METHOD PUBLIC M_Run : BOOL
VAR_INPUT
	run:bool; // set to true to run, false to stop;
END_VAR

this^.iq_stPFO.pv_xRunSW := run;
END_METHOD

END_FUNCTION_BLOCK

// POUs/Functions/Valves/functions/F_RoughPumpInlet_ILK
(*
	Determine whether a pump attached to the inlet of a roughing pump is safe to open. 
	
	Return true, signaling it is safe to open when the roughing pump is confirmed to be working. 
*)

FUNCTION F_RoughPumpInlet_ILK : BOOL
VAR_INPUT
	ScrollPump	:	ST_RoughPump;
END_VAR
VAR
END_VAR


F_RoughPumpInlet_ILK := (ScrollPump.eState = pumpRUNNING); (* Confirm that the roughing pump is running before opening the valve *)

END_FUNCTION

// POUs/Functions/Valves/functions/F_TURBO_VRC_ILK
(* Close the vic if the roughing pump pirani loses its at-vac setpoint while the turbo is pumping *)
FUNCTION F_TURBO_VRC_ILK : BOOL
VAR_INPUT

	i_xHiVac 	: BOOL;
	i_xRunPTM	: BOOL;
	i_xFLVac	: BOOL;

END_VAR
VAR

	rHysterisis : REAL := 0;

	xInterlock: BOOL;
	rTolerance: REAL := 20;
END_VAR

(* Close the vic if the roughing pump pirani loses its at-vac setpoint while the turbo is pumping *)
F_TURBO_VRC_ILK := (NOT i_xHiVac AND NOT i_xRunPTM AND NOT i_xFLVac) OR
					(NOT i_xRunPTM AND i_xFLVac) OR
					(i_xRunPTM AND i_xFLVac);

END_FUNCTION

// POUs/Functions/Valves/functions/F_TurboGateValve_ILK
(* This Function Block evaluates the ILK condition of the Turbo Gate valve *)
(* The logic Protects the Turbo pump from inlet pressure above the SP*)

FUNCTION F_TurboGateValve_ILK : BOOL (* function return TRUE when ILK is OK*)
VAR_INPUT
	i_Turbo : ST_PTM; // Turbo Pump
	i_stISG : ST_VG; //Gauge measuring inlet Pressure e.g Pirani
END_VAR
VAR
END_VAR

(* This Function Block evaluates the ILK condition of the Turbo Gate valve *)
(* The logic Protects the Turbo pump from inlet pressure above the SP*)
F_TurboGateValve_ILK := (NOT (i_Turbo.eState = pumpSTOPPED) AND NOT (i_Turbo.eState = pumpSTOPPING) AND NOT (i_Turbo.eState = pumpFAULT))
						AND (i_stISG.xPRESS_OK AND i_stISG.rPRESS < i_Turbo.rInletPressureSP);

END_FUNCTION

// POUs/Functions/Valves/functions/F_TurboGateValve_ILK_1
(* This Function Block evaluates the ILK condition of the Turbo Gate valve *)
(* The logic Protects the Turbo pump from inlet pressure above the SP*)

FUNCTION F_TurboGateValve_ILK_1 : BOOL (* function return TRUE when ILK is OK*)
VAR_INPUT
	i_Turbo : ST_PTM; // Turbo Pump
	i_stISG : ST_VG; //Gauge measuring inlet Pressure e.g Pirani
END_VAR
VAR
END_VAR

(* This Function Block evaluates the ILK condition of the Turbo Gate valve *)
(* The logic Protects the Turbo pump from inlet pressure above the SP*)
F_TurboGateValve_ILK_1 := (NOT (i_Turbo.eState = pumpSTOPPED) AND NOT (i_Turbo.eState = pumpFAULT))
						AND (i_stISG.xPRESS_OK AND i_stISG.rPRESS < i_Turbo.rInletPressureSP);

END_FUNCTION

// POUs/Functions/Valves/functions/F_TurboGateValve_Protection_ILK
(* This Function Block evaluates the ILK condition of the Turbo Gate valve *)
(* The logic Protects the Turbo pump from inlet pressure above the SP*)
(* And Protects the Turbo pump from backing pressure above the SP*)
(* And Protects the Turbo pump in the case of backing pump not running*)

FUNCTION F_TurboGateValve_Protection_ILK : BOOL (* function return TRUE when ILK is OK*)
VAR_INPUT
	i_Turbo : ST_PTM; // Turbo Pump
	i_stISG : ST_VG; //Gauge measuring inlet Pressure e.g Pirani
	i_stBSG : ST_VG; //Gauge measuring backing Pressure e.g Pirani
	ScrollPump	:	ST_RoughPump; // Roughing pump
END_VAR
VAR
END_VAR

(* This Function Block evaluates the ILK condition of the Turbo Gate valve *)
(* The logic Protects the Turbo pump from inlet pressure above the SP*)
F_TurboGateValve_Protection_ILK := (NOT (i_Turbo.eState = pumpSTOPPED) AND NOT (i_Turbo.eState = pumpSTOPPING) AND NOT (i_Turbo.eState = pumpFAULT))
						AND (i_stISG.xPRESS_OK AND i_stISG.rPRESS < i_Turbo.rInletPressureSP)
						AND (i_stBSG.xPRESS_OK AND i_stBSG.rPRESS < i_Turbo.rBackingPressureSP)
						AND (ScrollPump.eState = pumpRUNNING);

END_FUNCTION

// POUs/Functions/Valves/functions/F_VALVE_REL_ILK
(* OK, this is going to be a general-use function that will return whether the ratio of the pressures given is less than x orders of magnitude.
True iff 10^(-x) < a/b < 10^x.  Simple, right?  Just make sure it gets a positive order of magnitude and the pressures aren't 0. ~Scott *)   
{attribute 'no_check'}
FUNCTION F_VALVE_REL_ILK : BOOL
VAR_INPUT
	i_stUSG	:	ST_VG; // Upstream Gague
	i_stDSG	:	ST_VG; // Downstream Gague
	//Orders of magnitude allowed between up/downstream pressures for valve to open. Must be real positive integer.
	i_iOrdersMagnitude: INT;
END_VAR
VAR
	rPressRatio : REAL;
	rMaxRatioAllowed	:	LREAL := EXPT(10,i_iOrdersMagnitude);
	rMinRatioAllowed	:	LREAL := EXPT(10,(-i_iOrdersMagnitude));
END_VAR

(* S. Stubbs 11/2015 *)

(* OK, this is going to be a general-use function that will return whether the ratio of the pressures given is less than x orders of magnitude.
True iff 10^(-x) < a/b < 10^x.  Simple, right?  Just make sure it gets a positive order of magnitude and the pressures aren't 0. ~Scott *)   

(* Find ratio *)

IF i_stDSG.rPRESS <> 0 THEN
	rPressRatio := i_stUSG.rPRESS / i_stDSG.rPRESS;

	F_VALVE_REL_ILK := rPressRatio < rMaxRatioAllowed AND rMinRatioAllowed < rPressRatio;
ELSE
	F_VALVE_REL_ILK := FALSE;
END_IF

END_FUNCTION

// POUs/Functions/Valves/functions/F_VRC_DIODE_ILK
(* The principle is simple, a VRC should never open when B side pressure is greater than 
the A side pressure. *)

FUNCTION F_VRC_DIODE_ILK : BOOL
VAR_INPUT

	i_stPGA : ST_VG; // A side pressure gauge
	i_stPGB	: ST_VG; // B side pressure gauge

END_VAR
VAR

	rHysterisis : REAL := 0;

	xInterlock: BOOL;
	rTolerance: REAL := 20;
END_VAR

(* The principle is simple, a VRC should never open when B side pressure is greater than the A side pressure. *)
rTolerance := 20;
F_VRC_DIODE_ILK := ((i_stPGA.rPRESS + rTolerance >= i_stPGB.rPRESS + rHysterisis) OR i_stPGA.xBAKEOUT) AND i_stPGA.xPRESS_OK AND i_stPGB.xPRESS_OK;

(* OK it gets a bit more complicated with hysterisis,

Now, if the F_VIC_DIODE_ILK is FALSE then some hysterisis is added to the B side. But if it's OK then we just stick with making sure that the A side is greater than the B side

*)
(*
IF NOT F_VIC_DIODE_ILK THEN
Hysterisis := 40;
ELSE
Hysterisis := 0;
END_IF
*)

END_FUNCTION

// POUs/Functions/Valves/functions/F_VRC_DIODE_ILK_OK
(*The function returns TRUE i.e. ILK_OK when pressure on A side is greater than or equal to the pressure on B side*)
FUNCTION F_VRC_DIODE_ILK_OK : BOOL
VAR_INPUT

	i_stPGA : ST_VG; // A side pressure gauge
	i_stPGB	: ST_VG; // B side pressure gauge

END_VAR
VAR
	rHysterisis : REAL := 0;

	xInterlock: BOOL;
	rTolerance: REAL := 0;
END_VAR

(* The principle is simple, a VRC should never open when B side pressure is greater than the A side pressure. *)
F_VRC_DIODE_ILK_OK := (i_stPGA.rPRESS + rTolerance >= i_stPGB.rPRESS + rHysterisis) AND i_stPGA.xPRESS_OK AND i_stPGB.xPRESS_OK;

END_FUNCTION

// POUs/Functions/Valves/Interfaces/FB_TVGC_ADS
(* This function block is created for interface devices between different PLC*)
(* Not all the fields in the original structure is required, just few signals *)
(*Use with FB_ADS_WATCHDOG on remotePLC*)
FUNCTION_BLOCK FB_TVGC_ADS extends FB_ADS
VAR_INPUT
	sNetId : String; //NetID of the Destination PLC controller
	nPort : UINT; // port number
	sVarName : string;// the variable name of the (device) declared function block.
	iWatchdog:UDINT;//The watchdog variable name written to by the remote plc
END_VAR
VAR_OUTPUT
	{attribute 'pytmc' := 'pv: '}
	VGC:ST_VGC;
	bError:BOOL;
END_VAR
VAR
	fb_CheckWatchdog: FB_CheckWatchdog;
	fb_Read_VGC: FB_ReadAdsSymByName;
	ftReset: F_TRIG;
	xFirstPass: bool:= true;
END_VAR

ftReset(CLK:= fb_Read_VGC.bBusy OR xFirstPass);
xFirstPass:=false;
(*calling ADS read function*)
fb_Read_VGC(
	bRead:= ftReset.Q, 
	sNetId:= sNetId, 
	nPort:= nPort, 
	sVarName:= CONCAT(sVarName,'.iq_stValve'), 
	nDestAddr:= ADR(VGC), 
	nLen:= SIZEOF(VGC), 
	tTimeout:= , 
	eComMode:= eAdsComModeFastCom, 
	bBusy=> , 
	bError=> , 
	nErrorId=> );
	

(*Error*)
fb_CheckWatchdog(
	bEnable:= TRUE, 
	tWatchdogTime:= T#900ms, 
	nCnt:= iWatchdog , 
	bWatchdog=> , 
	nLastCnt=> );
bError:= fb_Read_VGC.bError OR fb_CheckWatchdog.bWatchdog;

ACT_Logger();

ACTION ACT_Logger:
IF tErrorPresent.Q THEN
 IF(fb_Read_VGC.bError) THEN fbLogger(sMsg:='ADS Read Error', eSevr:=TcEventSeverity.Critical); END_IF;
 IF(fb_CheckWatchdog.bWatchdog) THEN fbLogger(sMsg:='ADS Watchdog Error', eSevr:=TcEventSeverity.Critical); END_IF;
END_IF
END_ACTION

END_FUNCTION_BLOCK

// POUs/Functions/Valves/Interfaces/FB_Valve_Interface
(* This function block is created for interface devices between different PLC*)
(* Not all the fields in the original structure is required, just few signals *)
(* They have to be linked to the custom created variables on the EL6692/5 primary side*)

FUNCTION_BLOCK FB_Valve_Interface
VAR_INPUT
END_VAR
VAR_OUTPUT
	{attribute 'pytmc' := 'pv: '}
	VGC:ST_VGC;
END_VAR
VAR
	i_xOpnLS AT%I*	: BOOL;
	i_xClsLS AT%I*	: BOOL;
END_VAR

(* This function block is created for interface devices between different PLC*)
(* Not all the fields in the original structure is required, just few signals *)
(* They have to be linked to the custom created variables on the EL6692/5 primary side*)


VGC.i_xClsLS := i_xClsLS;
VGC.i_xOpnLS := i_xOpnLS;

END_FUNCTION_BLOCK

// POUs/Functions/Valves/Interfaces/FB_VFS_Interface
(*Used as soft IO mapping to create a psuedo valve to communicate over two task on the same PLC.*) 
(*for FAST shutter control*)
FUNCTION_BLOCK FB_VFS_Interface EXTENDS FB_Valve
VAR_INPUT
	IG : ST_VG; // The MKS422 Cold Cathode Data Structure
END_VAR
VAR_OUTPUT
	{attribute 'pytmc' := '
    pv: ;
    '}
	iq_stValve : ST_VFS; (* All valve data and states will be in this struct*)
	i_xVAC_FAULT_OK AT%I*: BOOL; (*Valve Vacuum OK, is set to False when there is Vacuum Fault*)
END_VAR
VAR
	
	tonOvrd	:	TON;
	tOvrd	:	TIME := T#10s;
	(*outputs*)
	q_xPRESS_OK AT%Q*: BOOL;
	q_xOPN_SW AT%Q*:BOOL;
	q_xCLS_SW AT%Q*:BOOL; (*external open signal e.g epics*)
	q_xVAC_FAULT_Reset AT%Q*: BOOL; (*Valve Vacuum OK, is set to False when there is Vacuum Fault*)
	q_xOverrideMode AT%Q*: BOOL; (*To be linked to global override bit. This Overrides Vacuum logic only, EPS, MPS and PMPS are still enforces*)
	q_xOverrideOpen AT%Q*: BOOL;
	
	(*inputs*)
	i_xTrigger AT %I* : BOOL;
	i_xVFS_Open AT %I* : BOOL;
	i_xVFS_Closed AT %I* : BOOL;
	{attribute 'pytmc' := '
    pv: MPS_FAULT_OK
	field: ZNAM MPS FAULT ;
	field: ONAM MPS OK ;
	io: i ;
	'}
	i_xMPS_OK AT%I*: BOOL;(*MPS Fault OK, is set when the Valve is Open and there is no trigger*)
	i_eVFS_State AT%I*: E_VGC; (*Interface*)
END_VAR

(*soft IO Mapping*)

q_xPRESS_OK := IG.xPRESS_OK;

(* Soft IO Mapping*)
IO();
///Check valve postion
IF iq_stValve.i_xClsLS AND  iq_stValve.i_xOpnLS THEN
	iq_stValve.eState:=INVALID;
ELSIF NOT iq_stValve.i_xClsLS AND iq_stValve.i_xOpnLS THEN 
	iq_stValve.eState:=OPEN;
ELSIF iq_stValve.i_xClsLS AND NOT iq_stValve.i_xOpnLS THEN 
	iq_stValve.eState:=CLOSED;
ELSIF NOT iq_stValve.i_xClsLS AND NOT iq_stValve.i_xOpnLS THEN 
	iq_stValve.eState:=MOVING;
ELSE
	iq_stValve.eState:=INVALID;
END_IF
//Override timer
tonOvrd(IN:=q_xOverrideOpen, PT:=tOvrd);
(* Soft IO Mapping*)
IO();
(*Logger*)
ACT_Logger();

ACTION ACT_Logger:
// ILK logger

IF i_xTrigger AND ePrevState = OPEN THEN
 		fbLogger(sMsg:='Fast valve triggered to close', eSevr:=TcEventSeverity.Critical);  	
END_IF


//STATE Logger  

IF ePrevState <> iq_stValve.eState THEN
	  CASE iq_stValve.eState OF
		INVALID:
			fbLogger(sMsg:='Valve invalid position.', eSevr:=TcEventSeverity.Critical);
  		MOVING:
			fbLogger(sMsg:='Valve moving', eSevr:=TcEventSeverity.Warning);
		OPEN:
			fbLogger(sMsg:='Valve Open.', eSevr:=TcEventSeverity.Info);
		CLOSED:
			fbLogger(sMsg:='Valve closed.', eSevr:=TcEventSeverity.Info);
	  END_CASE
	  ePrevState := iq_stValve.eState;  
  END_IF
  


// Log valve timeouts
tErrorPresent(CLK:=iq_stValve.bErrorPresent);
IF tErrorPresent.Q THEN fbLogger(sMsg:=iq_stValve.sErrorMessage, eSevr:=TcEventSeverity.Warning); END_IF

// Log valve open
tAction(CLK:= iq_stValve.q_xOPN_DO);
IF tAction.Q THEN fbLogger(sMsg:='Valve commanded open', eSevr:=TcEventSeverity.Info); END_IF

// Log override mode enabled
tOverrideActivated(CLK:= (tonOvrd.Q AND q_xOverrideMode));
IF tOverrideActivated.Q THEN fbLogger(sMsg:='Valve override mode activated', eSevr:=TcEventSeverity.Warning); END_IF
END_ACTION

ACTION IO:
(*inputs*)
iq_stValve.i_xTrigger := i_xTrigger;
iq_stValve.i_xOpnLS := 	i_xVFS_Open;
iq_stValve.i_xClsLS:=	i_xVFS_Closed;
iq_stValve.eVGC_State := i_eVFS_State;
iq_stValve.i_xVAC_FAULT_OK:= i_xVAC_FAULT_OK;
(*output*)
q_xOPN_SW := iq_stValve.pv_xOPN_SW;
q_xCLS_SW:= iq_stValve.xCLS_SW;
q_xVAC_FAULT_Reset :=  iq_stValve.pv_xAlmRst;
q_xOverrideMode :=iq_stValve.xOverrideMode;
q_xOverrideOpen := iq_stValve.pv_xOvrdOpn ;
iq_stValve.sGFS := IG.sPath;

//reset the commands 
IF ( iq_stValve.i_xOpnLS) THEN iq_stValve.pv_xOPN_SW := FALSE; END_IF
IF ( iq_stValve.i_xClsLS) THEN iq_stValve.xCLS_SW := FALSE; END_IF
END_ACTION

END_FUNCTION_BLOCK

// POUs/Functions/Valves/Interfaces/ITF_Valve
INTERFACE ITF_Valve

END_INTERFACE

// POUs/Functions/Valves/FB_Kashiyama_VRC
(* Main Kashiyama gate valve permit to be open when:
		1. pump is NORMAL operating status, and
	    2. chamber pressure is below HighSP or pump is at LowSpeed state.
	it will close if chamber pressure is below than lowSP for 180s.	
*)
FUNCTION_BLOCK FB_Kashiyama_VRC
VAR_IN_OUT
	
END_VAR
VAR_OUTPUT
	{attribute 'pytmc' := ' pv:'}
	q_stValve : ST_VRC;
END_VAR
VAR_INPUT
	Pump : ST_KashiyamaDryPump;//Kashyiama pump
	i_xExtILK_OK : BOOL; //Connect to Interlock logic condition(e.g F_TURBO_VRC_ILK Function), otherwise, Set to True if the valve is not interlocked
	Gauge : ST_VG;// Pressure Gauge	
	i_xOverrideMode : BOOL;
END_VAR
VAR
	At_HiVac : BOOL;
	tmrTP : TP;
	tmrPT: TIME := T#180S;
	v1: BOOL;
	tonOvrd	:	TON;
	tonDelOK : TON;
	rtOK	:	R_TRIG;
	
	(*IO*)
	i_xOpnLS	AT%I*: BOOL;
	i_xClsLS	AT%I*: BOOL;
	q_xOPN_DO	AT%Q*: BOOL;
	
END_VAR

(* Main Kashiyama gate valve permit to be open when:
		1. pump is NORMAL operating status, and
	    2. chamber pressure is below HighSP or pump is at LowSpeed state.
	it will close if chamber pressure is below than lowSP for 60s.	
*)
(* 
      For main Kayshiyama pump's gate valve:
		Pump LowSP is MU100 base pressure (20 mTorr) 
		Pump HighSP is 600 Torr;
	  Second Kayshiyama pump allow Gas Attenuator operating at higher pressure, 
      it's gate valve is to be open when Gas Attenuator chamber pressure is above lowSP.  
*)


///Check valve postion
IF NOT q_stValve.i_xClsLS AND q_stValve.i_xOpnLS THEN 
	q_stValve.eState:=OPEN;
ELSIF q_stValve.i_xClsLS AND NOT q_stValve.i_xOpnLS THEN 
	q_stValve.eState:=CLOSED;
ELSIF NOT q_stValve.i_xClsLS AND NOT q_stValve.i_xOpnLS THEN 
	q_stValve.eState:=MOVING;
ELSE
	q_stValve.eState:=INVALID;
END_IF

//valve open interlock
q_stValve.xOPN_OK := Pump.i_xIsRun AND Pump.RdyTmr <= 0.0 AND (Gauge.rPRESS < Pump.HighSP OR Pump.q_xLspdDo) AND i_xExtILK_OK;
 

(* Override logic *)
(* Goal: give ability to override, but do so in a way that people won't forget it.
Solution: Override only after ten seconds of override, protect against blips,
when the valve permission goes true for more than ten seconds consistently, remove override
*)

tonDelOK(IN:=q_stValve.xOPN_OK, PT:=T#10S);
rtOK(CLK:=tonDelOK.Q);
IF rtOK.Q THEN q_stValve.pv_xOvrdOpn :=FALSE; END_IF

//Override timer
tonOvrd(IN:=q_stValve.pv_xOvrdOpn, PT:=T#10S);


(* Here's where the valve closes *)
IF NOT q_stValve.xOPN_OK AND NOT tonOvrd.Q THEN
q_stValve.pv_xOPN_SW := FALSE;
END_IF

At_HiVac := Gauge.xPRESS_OK AND Gauge.rPRESS < Pump.LowSP;
tmrTP (IN := At_HiVac AND q_stValve.q_xOPN_DO , PT := tmrPT);

IF At_HiVac AND q_stValve.q_xOPN_DO AND NOT tmrTP.Q THEN
	q_stValve.pv_xOPN_SW := FALSE ;
END_IF

(* Here's where the valve opens *)
q_stValve.q_xOPN_DO := (q_stValve.pv_xOPN_SW AND q_stValve.xOPN_OK) OR (tonOvrd.Q AND i_xOverrideMode); 

(*Soft IO Mapping*)
ACT_IO();

ACTION ACT_IO:
(*inputs*)
q_stValve.i_xOpnLS := 	i_xOpnLS;
q_stValve.i_xClsLS:=	i_xClsLS;
(*outputs*)
q_xOPN_DO:= q_stValve.q_xOPN_DO;
END_ACTION

END_FUNCTION_BLOCK

// POUs/Functions/Valves/FB_MKS248
(* MKS248 valve using MKS1249 Drive Module *)
FUNCTION_BLOCK FB_MKS248
VAR_INPUT
	i_xExtIlkOK	:	BOOL; //External Interlock, SET to TRUE if not used
	i_rReqPos	:	REAL; //Requested position
END_VAR
VAR_OUTPUT
	{attribute 'pytmc' := 'pv:'}
	iq_stVFN	:	ST_VCN; //Needle valve structure
END_VAR
VAR CONSTANT
	rOpenVoltage	:	REAL := 9.8; 
	rCloseVoltage	:	REAL := 0;	
END_VAR
VAR
	// Requested voltage
	rReqVoltage: REAL := 0;
	(*IO*)
	q_iRawPosition AT%Q* :INT;
END_VAR

(* MKS248 valve using MKS1249 Drive Module *)


// Interlocking
iq_stVFN.xIlkOK := i_xExtIlkOK;
(*Checking which Control mode is selected*)
IF iq_stVFN.xIlkOK THEN
	IF iq_stVFN.eValveControl = OpenValve THEN
		iq_stVFN.rReqPosition := iq_stVFN.rUpperLimit;(*Percentage*)// iq_stVCN.rUpperLimit;
	ELSIF iq_stVFN.eValveControl = CloseValve THEN
		iq_stVFN.rReqPosition := 0; (*Percentage*)
	ELSIF iq_stVFN.eValveControl = ManualControl THEN
		iq_stVFN.rReqPosition := LIMIT(0, iq_stVFN.rReqPosition, iq_stVFN.rUpperLimit);
	ELSIF iq_stVFN.eValveControl = PressureControl THEN
		iq_stVFN.rReqPosition := LIMIT(0, i_rReqPos, iq_stVFN.rUpperLimit); 
	END_IF
ELSE
	iq_stVFN.rReqPosition := 0;
	iq_stVFN.eValveControl := CloseValve;
END_IF

// Requested Voltage calculation
rReqVoltage := iq_stVFN.rReqPosition * (rOpenVoltage-rCloseVoltage)/100 + rCloseVoltage;
rReqVoltage := LIMIT(rCloseVoltage, rReqVoltage, rOpenVoltage); //The requested voltage should remain within this range
//Raw position calc
iq_stVFN.q_iRawPosition := REAL_TO_INT( 32767/10 * rReqVoltage);	
(*IO Mapping*)
ACT_IO();

ACTION ACT_IO:
(*outputs*)
q_iRawPosition := iq_stVFN.q_iRawPosition;
END_ACTION

END_FUNCTION_BLOCK

// POUs/Functions/Valves/FB_TurbVentvalve_NO
(* This function block impelemets Interlock for Agilent Turbo Vent Valve Normally Open*)
FUNCTION_BLOCK FB_TurbVentvalve_NO
VAR_OUTPUT
	{attribute 'pytmc' :=' pv:'}
	q_stValve : ST_VCC_NO;
END_VAR
VAR_INPUT
	i_stPTM	: ST_AgilentPTM; //Agilent Turbo Pump
END_VAR
VAR
	tofTmr 		: 	TOF;
	
	(*Output*)
	q_xCLS_DO AT%Q* : BOOL;
END_VAR

(*If the turbo is on, you cannot open the valve. In order to open the valve, you have to allow the turbopump
 to have already been turned off for 2 minutes and you have to press the open button on the vent valve

If the code looks confusing please use a truth table to verify*)

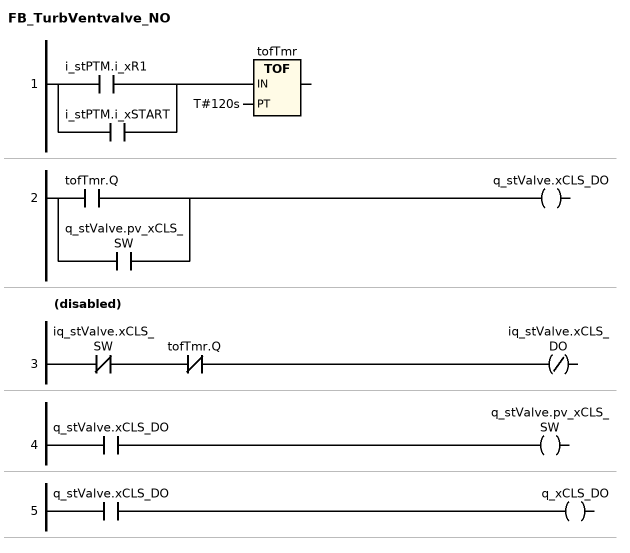
// NETWORK 1
tofTmr(IN := i_stPTM.i_xR1 OR i_stPTM.i_xSTART, PT := T#120s); // TOF

// NETWORK 2
q_stValve.xCLS_DO := tofTmr.Q OR q_stValve.pv_xCLS_SW;

// NETWORK 3 (disabled)
// iq_stValve.xCLS_DO := NOT (NOT iq_stValve.xCLS_SW AND NOT tofTmr.Q);

// NETWORK 4
q_stValve.pv_xCLS_SW := q_stValve.xCLS_DO;

// NETWORK 5
q_xCLS_DO := q_stValve.xCLS_DO;

ACTION ACT_IO:
(*outputs*)
q_xCLS_DO:= q_stValve.xCLS_DO;
END_ACTION

METHOD M_Close : BOOL
VAR_INPUT
		close:BOOL; //True to CLose, False to OPEN
END_VAR
This^.q_stValve.pv_xCLS_SW :=Close;
END_METHOD

END_FUNCTION_BLOCK

// POUs/Functions/Valves/FB_VCN
(* This function implements the Basic functions for the Pfeiffer EVR 116 needle valve*)
FUNCTION_BLOCK FB_VCN
VAR_INPUT
	i_xExtIlkOK	:	BOOL; //External Interlock, SET to TRUE if not used
	i_ReqPos	:	REAL; //Requested position

END_VAR
VAR_OUTPUT
	{attribute 'pytmc' := '
    pv:
	'}
	iq_stVCN	:	ST_VCN; //Needle valve structure
END_VAR
VAR_IN_OUT
	
END_VAR

VAR CONSTANT
	rOpenVoltage	:	REAL := 9.1; // From the EVR 116 manual, A Voltage of 9V it is completely Open
	rCloseVoltage	:	REAL := 0.4;// a voltage <0.5 V the valve is closed	
END_VAR
VAR
	// Requested voltage
	{attribute 'pytmc' := '
	pv: POS_AO;
	io: i ;
	'}
	rReqVoltage: REAL := 0;
	//iResolution: INT :=16;
	// 
	(*IO*)
	q_iRawPosition AT%Q* :INT;

END_VAR

(* Needle valve control FB
A. Wallace 2016-7-21

This FB should be used as a low level control block.

It provides:

Valve position ceiling
Interlock
Scaling

It is not intended for:
Closed-loop control

It could be used for:
Valve position/flow linearization

Note: Raw position calc is based on 0.5 to 9V span, 32767 bits
*)

// Interlocking
iq_stVCN.xIlkOK := i_xExtIlkOK;
(*Checking which Control mode is selected*)
IF iq_stVCN.xIlkOK THEN
	IF iq_stVCN.eValveControl = OpenValve THEN
		iq_stVCN.rReqPosition := iq_stVCN.rUpperLimit;(*Percentage*)// iq_stVCN.rUpperLimit;
	ELSIF iq_stVCN.eValveControl = CloseValve THEN
		iq_stVCN.rReqPosition := 0; (*Percentage*)
	ELSIF (iq_stVCN.eValveControl = ManualControl) (*AND (iq_stVCN.xOPN_SW)*) THEN
		iq_stVCN.rReqPosition := LIMIT(0, iq_stVCN.rReqPosition, iq_stVCN.rUpperLimit);
	ELSIF iq_stVCN.eValveControl = PressureControl THEN
		iq_stVCN.rReqPosition := LIMIT(0, i_ReqPos, iq_stVCN.rUpperLimit); 
	END_IF
ELSE
	iq_stVCN.rReqPosition := 0;
	iq_stVCN.eValveControl := CloseValve;
END_IF

// Requested Voltage calculation
rReqVoltage := iq_stVCN.rReqPosition * (rOpenVoltage-rCloseVoltage)/100 + rCloseVoltage;
rReqVoltage := LIMIT(rCloseVoltage, rReqVoltage, rOpenVoltage); //The requested voltage should remain within this range
//Raw position calc
iq_stvcn.q_iRawPosition := REAL_TO_INT( 32767/10 * rReqVoltage);	

(*SOft IO Mapping*)
ACT_IO();

ACTION ACT_IO:
(*outputs*)
q_iRawPosition := iq_stVCN.q_iRawPosition;
(*inputs*)
iq_stVCN.i_iPosition := iq_stvcn.q_iRawPosition;
END_ACTION

METHOD M_ValveControl : BOOL
VAR_INPUT
	state:E_VCN; // Close, Open, Pressure, Manual
END_VAR
iq_stVCN.eValveControl := state;
END_METHOD

END_FUNCTION_BLOCK

// POUs/Functions/Valves/FB_VFS
(* This function block implements basic functionality for Fast Shutter/Valves*)
(* Create a separate virtual PLC for the fast shutter logic, and tie/map this task to the FAST I/O portion of the ethercat bus,
 so we can scan these I/Os faster than the rest of the vacuum I/Os.
The Fast shutter was tested with PLC task Cycle Base Time 50us with cycle time 0.050ms.
*)
FUNCTION_BLOCK FB_VFS EXTENDS FB_Valve
VAR_INPUT
	i_xPMPS_OK:	BOOL	; (*External MPS interlock, Set to TRUE when no PMPS interlock is required*)
	i_xExt_OK: BOOL; (*Other External Interlock, Set to True when no external interlock is required*)
	i_sDevName : T_MaxString :=  'VGC'; // Device name for diagnostic
END_VAR
VAR_IN_OUT
	io_fbFFHWO    :    FB_HardwareFFOutput;
END_VAR
VAR
	xOPN_OK :BOOL;
	xERR_ExtFault :BOOL; 
	// PMPS
	fbFF    :    FB_FastFault :=(
        i_DevName := 'VFS',
        i_Desc := 'Fault occurs when fast valve is not in open state',
        i_TypeCode := 16#1010);
	
	rDiffPressAllowed	:	REAL := 22.5; // Torr, Default value comes from Vat Valve Manual
	rDiffPress : REAL;
	set : BOOL;
    reset: BOOL;
	  
	xFirstPass	:	BOOL := TRUE;
	//fbFSInit		:	R_TRIG;
	rtOPN_SW :	R_TRIG;
		
	tonDelOK : TON;
	rtOK	:	R_TRIG;
	tonOvrd	:	TON;
	
	tDelOK	:	TIME := T#60S;
	tOvrd	:	TIME := T#10s;
	
	xClose: BOOL;
	xOpen: BOOL;
	CloseTimer: TON;
	TimDur: TIME := T#20MS;
	OpenTimer: TON;
	OpenTimDur: TIME := T#2S;
	
	(* Timeouts*)
	tCLSTimeOutDuration: TIME:= T#0.5S;
	tOPNTimeOutDuration: TIME:= T#10S;
	tOPNtimeout: TON;
	tCLStimeout:TON;
	

	(*IO*)
	i_xOpnLS	AT%I*: BOOL;
	i_xClsLS	AT%I*: BOOL;
	q_xClose_A	AT%Q*: BOOL;
	q_xClose_B	AT%Q*: BOOL;
	q_xClose_C	AT%Q*: BOOL;
	q_xOPN_DO	AT%Q*: BOOL;
	i_xTrigger	AT%I*: BOOL; 
	
	// Interface
	i_xPress_OK AT%I*:BOOL; (*To be linked to the Fast sensor structure signal IG.xPRESS_OK, to make sure that the device is connected*)
	i_xOPN_SW AT%I*:BOOL;
	i_xCLS_SW AT%I*:BOOL; (*external open signal e.g epics*)
	i_xVAC_FAULT_Reset	AT%I*: BOOL;(*Valve Vacuum OK, is set to False when there is Vacuum Fault*)
	i_xOverrideMode AT%I*: BOOL; (*To be linked to global override bit. This Overrides Vacuum logic only, EPS, MPS and PMPS are still enforces*)
	i_xOverrideOpen AT%I*: BOOL;
	q_xTrigger	AT%Q*: BOOL; (*Interface*)
	q_xVFS_Open AT%Q*: BOOL; (*Interface*)
	q_xVFS_Closed AT%Q*: BOOL; (*Interface*)
	q_xVAC_FAULT_OK AT%Q*: BOOL; (*Valve Vacuum OK, is set to False when there is Vacuum Fault*)
	q_xMPS_OK	 AT%Q*:	BOOL; (*MPS Fault OK, is set when the Valve is Open and there is no trigger*)
	q_eVFS_State AT%Q*: E_VGC; (*Interface*)
	
END_VAR



(* Fast Shutter/Valve Function Block*)
(* M.Ghaly Feb 2019*)

(* Fast Shutters do not function as complete isolation valves, but are intended to rapidly limit conductance 
between vacuum regions.  They should be installed in conjunction with isolation gate valves.  The conductance 
of the fast shutter in the closed state may be sufficiently low as to create an isolated vacuum region.  
Thus, at least a pirani gauge, that can measure a pressure down to 1x10-4 Torr, needs to be installed between
the shutter and the isolation gate valve.
In the case where a gauge is not installed, the neigboring gate Valves should not be opened unless the shutter 
is Open. 
*)
(* On first PLC pass, put valve into vented state, which implies a closed valve *)
IF xFirstPass THEN
	fbFF.i_DevName := i_sDevName;
	xFirstPass := FALSE;
END_IF

(* Input Trigger to close the Fast Shutter*)
(* Neighboring Valves Should also be triggered to Close*)
IF (i_xTrigger) OR NOT (i_xPress_OK) OR NOT (i_xExt_OK)  OR i_xCLS_SW  THEN 
	xClose:= TRUE;
	xOpen:= FALSE;
	q_xVAC_FAULT_OK:= FALSE;
	IF (NOT i_xCLS_SW) THEN xERR_ExtFault := TRUE; END_IF;
	i_xCLS_SW := TRUE;
	q_xOPN_DO := FALSE;
	//i_xOPN_SW :=FALSE;
	xOpen:=FALSE;
ELSIF ((rtOPN_SW.Q) AND xOPN_OK AND NOT i_xOpnLS) OR (tonOvrd.Q AND i_xOverrideMode) THEN
	q_xOPN_DO := TRUE;
END_IF
IF (xClose) AND (NOT i_xClsLS) THEN
	q_xClose_A := TRUE;
	q_xClose_B := TRUE;
	q_xClose_C := TRUE;
END_IF
IF(CloseTimer.Q) OR (i_xClsLS) THEN
	q_xClose_A := FALSE;
	q_xClose_B := FALSE;
	q_xClose_C := FALSE;
	xClose := FALSE;
	//i_xOPN_SW := FALSE;
END_IF

IF(OpenTimer.Q) AND (i_xOpnLS) THEN
	q_xOPN_DO :=  FALSE;
	i_xOPN_SW := FALSE;
	xOpen:=FALSE;
END_IF

(* Neighboring Valves Interlock bit is reset When the Vacuum event error is reset and the Shutter is opened *)
IF (NOT i_xTrigger) AND (NOT xERR_ExtFault) AND i_xOpnLS THEN
	q_xVAC_FAULT_OK := TRUE;
END_IF

(*OPN OK evaluation bit *)
xOPN_OK := (NOT xERR_ExtFault) AND NOT i_xTrigger;

(* If Epics Command to close the Valve, check if PMPS, otherwise Keep command set to open valve *)
// is there really a PMPS requirment.



(* When the valve  is open MPS is OK*)
q_xMPS_OK := i_xOpnLS AND NOT i_xTrigger AND i_xPress_OK AND NOT(i_xCLS_SW);


(* Override logic *)
(* Goal: give ability to override, but do so in a way that people won't forget it.
Solution: Override only after ten seconds of override, protect against blips,
when the valve permission goes true for more than ten seconds consistently, remove override
*)

tonDelOK(IN:=xOPN_OK, PT:=tDelOK);
rtOK(CLK:=tonDelOK.Q);
IF rtOK.Q AND i_xOverrideOpen THEN 
	i_xOverrideOpen :=FALSE;
	//if (iq_stValve.eState = OPEN) AND (i_xOverrideMode) THEN iq_stValve.pv_xOPN_SW := TRUE; END_IF //for seamless transition   
    //Log
    fbLogger(sMsg:='Override expired', eSevr:=TcEventSeverity.Warning);
END_IF

//Override timer
tonOvrd(IN:=i_xOverrideOpen, PT:=tOvrd);


//Assign valve state
IF (i_xTrigger) THEN q_eVFS_State := E_VGC.Triggered;
ELSIF xERR_ExtFault THEN q_eVFS_State :=  E_VGC.Vac_Fault;
ELSIF NOT i_xClsLS AND tCLStimeout.Q THEN 
	q_eVFS_State :=  E_VGC.Cls_Timeout;
ELSIF NOT i_xOpnLS AND tOPNtimeout.Q THEN 
	q_eVFS_State :=  E_VGC.Opn_Timeout;
ELSE q_eVFS_State :=  E_VGC.At_Vac;
END_IF

(*Timers*)
CloseTimer ( IN:=xClose, PT:= TimDur, Q=>);
OpenTimer ( IN:=i_xOpnLS, PT:= OpenTimDur, Q=>);
tOPNtimeout(IN:= q_xOPN_DO, PT := tOPNTimeOutDuration);
tCLStimeout(IN:= q_xClose_A, PT := tCLSTimeOutDuration);
rtOPN_SW(CLK:= i_xOPN_SW);

(* Soft IO Mapping*)
IO();

(*Alarm reset *)
ACT_ResetAlarms();

(*FAST FAULT*)
fbFF(i_xOK := q_xMPS_OK,
    i_xReset := i_xVAC_FAULT_Reset,
	i_xAutoReset :=TRUE,
    io_fbFFHWO := io_fbFFHWO);

ACTION ACT_ResetAlarms:
//iq_stValve.xERR_DifPres R= i_xResetFault;

//iq_stValve.bErrorPresent R= i_xResetFault;

IF NOT i_xTrigger AND i_xPress_OK THEN
	xERR_ExtFault R= i_xVAC_FAULT_Reset;
	i_xVAC_FAULT_Reset:=FALSE;
END_IF
END_ACTION

ACTION IO:

q_xTrigger := i_xTrigger;
q_xVFS_Closed:= i_xClsLS;
q_xVFS_Open:= i_xOpnLS;
END_ACTION

END_FUNCTION_BLOCK

// POUs/Functions/Valves/FB_VRC
(* This Function Block Implements Basic Functionality for certain types of valves e.g Turbo Isolation valves, Apperture Valve.
This function block is interloked by an input (i_xExtILK_OK). This is so developers can interface with custom
interlocking logic outside this function block.*)
(* Note Interlock Logic is External *)
{attribute 'no_check'}
FUNCTION_BLOCK FB_VRC EXTENDS FB_Valve
VAR_IN_OUT
	
END_VAR
VAR_INPUT
	i_xExtILK_OK : BOOL; //Connect to Interlock logic condition(e.g F_TURBO_VRC_ILK Function), otherwise, Set to True if the valve is not interlocked
	i_xOverrideMode : BOOL; (*To be linked to global override bit. This Overrides Vacuum logic only, EPS, MPS and PMPS are still enforces*)
END_VAR
VAR_OUTPUT
	{attribute 'pytmc' := '
    pv:
	'}
	iq_stValve : ST_VRC;
END_VAR
VAR
	{attribute 'instance-path'}
	{attribute 'noinit'}
	sPath: STRING;
	xFirstPass	:	BOOL;
	fbFSInit		:	R_TRIG;
	tonOvrd	:	TON;
	tonDelOK : TON;
	rtOK	:	R_TRIG;
	tOvrd	:	TIME := T#10s;
	(* Timeouts*)
	tTimeOutDuration: TIME:= T#30S;
	tOPNtimeout: TON;
	tCLStimeout:TON;
	
	
	(*IO*)
	i_xOpnLS	AT%I*: BOOL;
	i_xClsLS	AT%I*: BOOL;
	q_xOPN_DO	AT%Q*: BOOL;

END_VAR


(* On first PLC pass, put valve into vented state, which implies a closed valve *)
fbFSInit( CLK := TRUE, Q => xFirstPass);
IF xFirstPass THEN
	iq_stValve.eVGC_State := Vented;
	iq_stValve.pv_xOPN_SW := FALSE;
	ePrevState := INVALID; 
END_IF




///Check valve position
IF iq_stValve.i_xClsLS AND  iq_stValve.i_xOpnLS THEN
	iq_stValve.eState:=INVALID;
ELSIF NOT iq_stValve.i_xClsLS AND iq_stValve.i_xOpnLS AND iq_stValve.q_xOPN_DO THEN 
	iq_stValve.eState:=OPEN;
ELSIF NOT iq_stValve.i_xClsLS AND iq_stValve.i_xOpnLS AND NOT iq_stValve.q_xOPN_DO THEN 
	iq_stValve.eState:=OPEN_F;
ELSIF iq_stValve.i_xClsLS AND NOT iq_stValve.i_xOpnLS AND NOT iq_stValve.q_xOPN_DO THEN 
	iq_stValve.eState:=CLOSED;
ELSIF NOT iq_stValve.i_xClsLS AND NOT iq_stValve.i_xOpnLS THEN 
	iq_stValve.eState:=MOVING;
ELSE
	iq_stValve.eState:=INVALID;
END_IF


(*evaluate Valve open external interlock*)
iq_stValve.xOPN_OK := i_xExtILK_OK;
iq_stValve.xEXT_OK := i_xExtILK_OK;
IF NOT iq_stValve.xOPN_OK and NOT tonOvrd.Q THEN
	iq_stValve.pv_xOPN_SW := FALSE;
	iq_stValve.eVGC_State := ERR_ExtFault;
END_IF

IF (iq_stValve.q_xOPN_DO) AND (iq_stValve.xOPN_OK) THEN
	iq_stValve.eVGC_State := AtVacuum;
END_IF
	

(* Override logic *)
(* Goal: give ability to override, but do so in a way that people won't forget it.
Solution: Override only after ten seconds of override, protect against blips,
when the valve permission goes true for more than ten seconds consistently, remove override
*)

tonDelOK(IN:=iq_stValve.xOPN_OK, PT:=T#10S);
rtOK(CLK:=tonDelOK.Q);
IF rtOK.Q AND iq_stValve.pv_xOvrdOpn THEN 
	iq_stValve.pv_xOvrdOpn :=FALSE; 
	if (iq_stValve.eState=OPEN) AND (i_xOverrideMode) THEN iq_stValve.pv_xOPN_SW := TRUE; END_IF
    //Log
    fbLogger(sMsg:='Override expired', eSevr:=TcEventSeverity.Warning);
END_IF
// Release the Force Open bit when the system override is false
IF NOT(i_xOverrideMode) THEN  iq_stValve.pv_xOvrdOpn :=FALSE; END_IF
//Override timer
tonOvrd(IN:=iq_stValve.pv_xOvrdOpn, PT:=tOvrd);

(* Here's where the valve opens *)
iq_stValve.q_xOPN_DO := (iq_stValve.pv_xOPN_SW AND iq_stValve.xOPN_OK) OR (tonOvrd.Q AND i_xOverrideMode);


///Check valve moving position timout
IF NOT iq_stValve.i_xClsLS AND tCLStimeout.Q THEN 
	iq_stValve.bErrorPresent := TRUE;
	iq_stValve.sErrorMessage := ' Close Timeout';
ELSIF NOT iq_stValve.i_xOpnLS AND tOPNtimeout.Q THEN 
	iq_stValve.bErrorPresent := TRUE; 
	iq_stValve.sErrorMessage := ' Open Timeout';
END_IF
IF (iq_stValve.eState=INVALID) THEN
	iq_stValve.bErrorPresent := TRUE; 
	iq_stValve.sErrorMessage := CONCAT(sPath,' Invalid Valve Position');
END_IF

(*Timers*)
tOPNtimeout(IN:= iq_stValve.q_xOPN_DO, PT := tTimeOutDuration );
tCLStimeout(IN:= NOT iq_stValve.q_xOPN_DO, PT := tTimeOutDuration);


(*Soft IO Mapping*)
ACT_IO();

// Log States and triggers
ACT_Logger();

ACTION ACT_IO:
(*inputs*)
iq_stValve.i_xOpnLS := 	i_xOpnLS;
iq_stValve.i_xClsLS:=	i_xClsLS;
iq_stValve.xOverrideMode := i_xOverrideMode;
(*outputs*)
q_xOPN_DO:= iq_stValve.q_xOPN_DO;
END_ACTION

ACTION ACT_Logger:
// ILK logger

IF NOT i_xExtILK_OK AND ePrevState = OPEN THEN
 		fbLogger(sMsg:='Lost external interlock while valve was open.', eSevr:=TcEventSeverity.Critical);  	
END_IF


//STATE Logger  

IF ePrevState <> iq_stValve.eState THEN
	  CASE iq_stValve.eState OF
		INVALID:
			fbLogger(sMsg:='Valve invalid position.', eSevr:=TcEventSeverity.Critical);
  		MOVING:
			fbLogger(sMsg:='Valve moving', eSevr:=TcEventSeverity.Warning);
		OPEN:
			fbLogger(sMsg:='Valve Open.', eSevr:=TcEventSeverity.Info);
		CLOSED:
			fbLogger(sMsg:='Valve closed.', eSevr:=TcEventSeverity.Info);
	  END_CASE
	  ePrevState := iq_stValve.eState;  
  END_IF
  


// Log valve timeouts
tErrorPresent(CLK:=iq_stValve.bErrorPresent);
IF tErrorPresent.Q THEN fbLogger(sMsg:=iq_stValve.sErrorMessage, eSevr:=TcEventSeverity.Warning); END_IF

// Log valve open
tAction(CLK:= iq_stValve.q_xOPN_DO);
IF tAction.Q THEN fbLogger(sMsg:='Valve commanded open', eSevr:=TcEventSeverity.Info); END_IF

// Log override mode enabled
tOverrideActivated(CLK:= (tonOvrd.Q AND i_xOverrideMode));
IF tOverrideActivated.Q THEN fbLogger(sMsg:='Valve override mode activated', eSevr:=TcEventSeverity.Warning); END_IF
END_ACTION

METHOD PUBLIC M_IsClosed : BOOL
VAR_INPUT
END_VAR
M_IsClosed := (This^.iq_stValve.eState = E_ValvePositionState.CLOSED);
END_METHOD

METHOD PUBLIC M_IsOpen : BOOL
VAR_INPUT
END_VAR
M_IsOpen := (This^.iq_stValve.eState = E_ValvePositionState.OPEN);
END_METHOD

// Use this Methode to Open or close the valve by setting the OPN_SW to the input value.
METHOD PUBLIC M_Set_OPN_SW : BOOL
VAR_INPUT
	value:BOOL;
END_VAR
This^.iq_stValve.pv_xOPN_SW := value;
END_METHOD

END_FUNCTION_BLOCK

// POUs/Functions/Valves/FB_VRC_EBD
(* This function block is similar to the FB_VGC, except it has 2 outputs to actuate the Valve*)
(* This Function Block Implements Basic Functionality for certain types of valves e.g Turbo Isolation valves, Apperture Valve *)
(* Note Interlock Logic is External *)
FUNCTION_BLOCK FB_VRC_EBD EXTENDS FB_Valve
VAR_IN_OUT
	
END_VAR
VAR_INPUT
	i_xExtILK_OK : BOOL; //Connect to Interlock logic condition(e.g F_TURBO_VRC_ILK Function), otherwise, Set to True if the valve is not interlocked
	i_xOverrideMode : BOOL; (*To be linked to global override bit. This Overrides Vacuum logic only, EPS, MPS and PMPS are still enforces*)
END_VAR
VAR_OUTPUT
	{attribute 'pytmc' := '
    pv:
	'}
	iq_stValve : ST_VRC;
END_VAR
VAR
	{attribute 'instance-path'}
	{attribute 'noinit'}
	sPath: STRING;
	xFirstPass	:	BOOL;
	fbFSInit		:	R_TRIG;
	tonOvrd	:	TON;
	tonDelOK : TON;
	rtOK	:	R_TRIG;
	tOvrd	:	TIME := T#10s;
	(* Timeouts*)
	tTimeOutDuration: TIME:= T#30S;
	tOPNtimeout: TON;
	tCLStimeout:TON;

	(*IO*)
	i_xOpnLS	AT%I*: BOOL;
	i_xClsLS	AT%I*: BOOL;
	q_xOPN_DO	AT%Q*: BOOL;
	q_xOPN_DO_2	AT%Q*: BOOL;
END_VAR


(* On first PLC pass, put valve into vented state, which implies a closed valve *)
fbFSInit( CLK := TRUE, Q => xFirstPass);
IF xFirstPass THEN
	iq_stValve.eVGC_State := Vented;
	iq_stValve.pv_xOPN_SW := FALSE;
END_IF


///Check valve position
IF NOT iq_stValve.i_xClsLS AND iq_stValve.i_xOpnLS THEN 
	iq_stValve.eState:=OPEN;
ELSIF iq_stValve.i_xClsLS AND NOT iq_stValve.i_xOpnLS THEN 
	iq_stValve.eState:=CLOSED;
ELSIF NOT iq_stValve.i_xClsLS AND NOT iq_stValve.i_xOpnLS THEN 
	iq_stValve.eState:=MOVING;
ELSE
	iq_stValve.eState:=INVALID;
END_IF

(*evaluate Valve open external interlock*)
iq_stValve.xOPN_OK := i_xExtILK_OK;
iq_stValve.xEXT_OK := i_xExtILK_OK;
IF NOT iq_stValve.xOPN_OK and NOT tonOvrd.Q THEN
	iq_stValve.pv_xOPN_SW := FALSE;
	iq_stValve.eVGC_State := ERR_ExtFault;
END_IF

IF (iq_stValve.q_xOPN_DO) AND (iq_stValve.xOPN_OK) THEN
	iq_stValve.eVGC_State := AtVacuum;
END_IF

(* Override logic *)
(* Goal: give ability to override, but do so in a way that people won't forget it.
Solution: Override only after ten seconds of override, protect against blips,
when the valve permission goes true for more than ten seconds consistently, remove override
*)

tonDelOK(IN:=iq_stValve.xOPN_OK, PT:=T#10S);
rtOK(CLK:=tonDelOK.Q);
IF rtOK.Q AND iq_stValve.pv_xOvrdOpn THEN 
	iq_stValve.pv_xOvrdOpn :=FALSE; 
	if (iq_stValve.eState=OPEN) AND (i_xOverrideMode) THEN iq_stValve.pv_xOPN_SW := TRUE; END_IF
    //Log
    fbLogger(sMsg:='Override expired', eSevr:=TcEventSeverity.Warning);
END_IF

//Override timer
tonOvrd(IN:=iq_stValve.pv_xOvrdOpn, PT:=T#10S);

(* Here's where the valve opens *)
iq_stValve.q_xOPN_DO := (iq_stValve.pv_xOPN_SW AND iq_stValve.xOPN_OK) OR (tonOvrd.Q AND i_xOverrideMode);

///Check valve moving postion timout
IF NOT iq_stValve.i_xClsLS AND tCLStimeout.Q THEN 
	iq_stValve.bErrorPresent := TRUE;
	iq_stValve.sErrorMessage := ' Close Timeout';
ELSIF NOT iq_stValve.i_xOpnLS AND tOPNtimeout.Q THEN 
	iq_stValve.bErrorPresent := TRUE; 
	iq_stValve.sErrorMessage := ' Open Timeout';
END_IF
IF (iq_stValve.eState=INVALID) THEN
	iq_stValve.bErrorPresent := TRUE; 
	iq_stValve.sErrorMessage := CONCAT(sPath,' Invalid Valve Position');
END_IF

(*Timers*)
tOPNtimeout(IN:= iq_stValve.q_xOPN_DO, PT := tTimeOutDuration );
tCLStimeout(IN:= NOT iq_stValve.q_xOPN_DO, PT := tTimeOutDuration);




(*Soft IO Mapping*)
ACT_IO();

// Log States and triggers
ACT_Logger();

ACTION ACT_IO:
(*inputs*)
iq_stValve.i_xOpnLS := 	i_xOpnLS;
iq_stValve.i_xClsLS:=	i_xClsLS;
iq_stValve.xOverrideMode := i_xOverrideMode;
(*outputs*)
q_xOPN_DO:= iq_stValve.q_xOPN_DO;
q_xOPN_DO_2:= iq_stValve.q_xOPN_DO;
END_ACTION

ACTION ACT_Logger:
// ILK logger

IF NOT i_xExtILK_OK AND ePrevState = OPEN THEN
 		fbLogger(sMsg:='Lost external interlock while valve was open.', eSevr:=TcEventSeverity.Critical);  	
END_IF


//STATE Logger  

IF ePrevState <> iq_stValve.eState THEN
	  CASE iq_stValve.eState OF
		INVALID:
			fbLogger(sMsg:='Valve invalid position.', eSevr:=TcEventSeverity.Critical);
  		MOVING:
			fbLogger(sMsg:='Valve moving', eSevr:=TcEventSeverity.Warning);
		OPEN:
			fbLogger(sMsg:='Valve Open.', eSevr:=TcEventSeverity.Info);
		CLOSED:
			fbLogger(sMsg:='Valve closed.', eSevr:=TcEventSeverity.Info);
	  END_CASE
	  ePrevState := iq_stValve.eState;  
  END_IF
  


// Log valve timeouts
tErrorPresent(CLK:=iq_stValve.bErrorPresent);
IF tErrorPresent.Q THEN fbLogger(sMsg:=iq_stValve.sErrorMessage, eSevr:=TcEventSeverity.Warning); END_IF

// Log valve open
tAction(CLK:= iq_stValve.q_xOPN_DO);
IF tAction.Q THEN fbLogger(sMsg:='Valve commanded open', eSevr:=TcEventSeverity.Info); END_IF

// Log override mode enabled
tOverrideActivated(CLK:= (tonOvrd.Q AND i_xOverrideMode));
IF tOverrideActivated.Q THEN fbLogger(sMsg:='Valve override mode activated', eSevr:=TcEventSeverity.Warning); END_IF
END_ACTION

METHOD PUBLIC M_IsClosed : BOOL
VAR_INPUT
END_VAR
M_IsClosed := (This^.iq_stValve.eState = E_ValvePositionState.CLOSED);
END_METHOD

METHOD PUBLIC M_IsOpen : BOOL
VAR_INPUT
END_VAR
M_IsOpen := (This^.iq_stValve.eState = E_ValvePositionState.OPEN);
END_METHOD

// Use this Methode to Open or close the valve by setting the OPN_SW to the input value.
METHOD PUBLIC M_Set_OPN_SW : BOOL
VAR_INPUT
	value:BOOL;
END_VAR
This^.iq_stValve.pv_xOPN_SW := value;
END_METHOD

END_FUNCTION_BLOCK

// POUs/Functions/Valves/FB_VRC_NO
(* This function block is different from the regular VRC in that CLOSING must be permitted. *)
FUNCTION_BLOCK FB_VRC_NO EXTENDS FB_Valve
VAR_IN_OUT

END_VAR
VAR_INPUT
	{attribute 'pytmc' := '
	pv: EXT_ILK_OK ;
	field: ZNAM NOT OK ;
	field: ONAM OK ;
	io: i ;
	'}
	i_xExtILK_OK : BOOL; //Connect to Interlock logic condition(e.g F_TURBO_VRC_ILK Function), otherwise, Set to True if the valve is not interlocked
	i_xOverrideMode : BOOL; (*To be linked to global override bit. This Overrides Vacuum logic only, EPS, MPS and PMPS are still enforces*)

END_VAR
VAR_OUTPUT
		iq_stValve : ST_VRC;
END_VAR
VAR

	{attribute 'noinit'}
	sPath: STRING;
	xFirstPass	:	BOOL;
	fbFSInit		:	R_TRIG;
	tonOvrd	:	TON;
	tonDelOK : TON;
	rtOK	:	R_TRIG;
	tOvrd	:	TIME := T#10s;
	(* Timeouts*)
	tTimeOutDuration: TIME:= T#30S;
	tOPNtimeout: TON;
	tCLStimeout:TON;
		{attribute 'pytmc' := '
	pv: CLS_SW ;
	field: ONAM CLOSE; 
	field: ZNAM OPEN;
	io: io ;
	'}
	pv_xCLS_SW	: BOOL;
	{attribute 'pytmc' := '
    pv: FORCE_CLS;
	io: io;
	'}
	pv_xOvrdCls	:	BOOL;

(*IO*)
	i_xOpnLS	AT%I*: BOOL;
	i_xClsLS	AT%I*: BOOL;
	q_xCLS_DO	AT%Q*: BOOL;

END_VAR

(* This function block is different from the regular VRC in that CLOSING must be permitted. *)

(* On first PLC pass, put valve into vented state, which implies a closed valve *)
fbFSInit( CLK := TRUE, Q => xFirstPass);
IF xFirstPass THEN
	pv_xCLS_SW := FALSE;
END_IF




///Check valve position
IF iq_stValve.i_xClsLS AND  iq_stValve.i_xOpnLS THEN
	iq_stValve.eState:=INVALID;
ELSIF NOT iq_stValve.i_xClsLS AND iq_stValve.i_xOpnLS AND iq_stValve.q_xOPN_DO THEN 
	iq_stValve.eState:=OPEN;
ELSIF iq_stValve.i_xClsLS AND NOT iq_stValve.i_xOpnLS AND NOT iq_stValve.q_xOPN_DO THEN 
	iq_stValve.eState:=CLOSED;
ELSIF NOT iq_stValve.i_xClsLS AND NOT iq_stValve.i_xOpnLS THEN 
	iq_stValve.eState:=MOVING;
ELSE
	iq_stValve.eState:=INVALID;
END_IF


(*evaluate Valve CLose external interlock*)
iq_stValve.xCLS_OK := i_xExtILK_OK;
IF NOT iq_stValve.xCLS_OK and NOT tonOvrd.Q THEN
	pv_xCLS_SW := FALSE;
END_IF


(* Override logic *)
(* Goal: give ability to override, but do so in a way that people won't forget it.
Solution: Override only after ten seconds of override, protect against blips,
when the valve permission goes true for more than ten seconds consistently, remove override
*)

tonDelOK(IN:=iq_stValve.xCLS_OK, PT:=T#10S);
rtOK(CLK:=tonDelOK.Q);
IF rtOK.Q AND pv_xOvrdCls THEN 
	pv_xOvrdCls :=FALSE; 
	if (iq_stValve.eState=CLOSED) AND (i_xOverrideMode) THEN pv_xCLS_SW := TRUE; END_IF
    //Log
    fbLogger(sMsg:='Override expired', eSevr:=TcEventSeverity.Warning);
END_IF

//Override timer
tonOvrd(IN:=pv_xOvrdCls, PT:=tOvrd);

(* Here's where the valve Actuates *)
q_xCLS_DO := ((iq_stValve.xCLS_OK  AND pv_xCLS_SW)OR (tonOvrd.Q AND i_xOverrideMode));
iq_stValve.q_xOPN_DO := NOT q_xCLS_DO;



///Check valve moving position timout
IF NOT iq_stValve.i_xClsLS AND tCLStimeout.Q THEN 
	iq_stValve.bErrorPresent := TRUE;
	//iq_stValve.sErrorMessage := ' Close Timeout';
ELSIF NOT iq_stValve.i_xOpnLS AND tOPNtimeout.Q THEN 
	iq_stValve.bErrorPresent := TRUE; 
	//iq_stValve.sErrorMessage := ' Open Timeout';
END_IF
IF (iq_stValve.eState=INVALID) THEN
	iq_stValve.bErrorPresent := TRUE; 
	//iq_stValve.sErrorMessage := CONCAT(sPath,' Invalid Valve Position');
END_IF

(*Timers*)
tOPNtimeout(IN:= iq_stValve.q_xOPN_DO, PT := tTimeOutDuration );
tCLStimeout(IN:= NOT iq_stValve.q_xOPN_DO, PT := tTimeOutDuration);


(*Soft IO Mapping*)
ACT_IO();

// Log States and triggers
ACT_Logger();

ACTION ACT_IO:
(*inputs*)
iq_stValve.i_xOpnLS := 	i_xOpnLS;
iq_stValve.i_xClsLS:=	i_xClsLS;
//iq_stValve. := i_xEXT_OK;
iq_stValve.xOverrideMode := i_xOverrideMode;
(*outputs*)
//q_xOPN_DO:= iq_stValve.q_xOPN_DO;
END_ACTION

METHOD PUBLIC M_IsClosed : BOOL
VAR_INPUT
END_VAR
M_IsClosed := (This^.iq_stValve.eState = E_ValvePositionState.CLOSED);
END_METHOD

METHOD PUBLIC M_IsOpen : BOOL
VAR_INPUT
END_VAR
M_IsOpen := (This^.iq_stValve.eState = E_ValvePositionState.OPEN);
END_METHOD

// Use this Methode to Open or close the valve by setting the OPN_SW to the input value.
METHOD PUBLIC M_Set_CLS_SW : BOOL
VAR_INPUT
		value:BOOL;
END_VAR
This^.pv_xCLS_SW := value;
END_METHOD

END_FUNCTION_BLOCK

// POUs/Functions/Valves/FB_VRC_OK_CLS
(* This function block is different from the regular VRC in that CLOSING must be permitted. *)
FUNCTION_BLOCK FB_VRC_OK_CLS
VAR_IN_OUT
	iq_stValve : ST_VRC;
END_VAR
VAR_INPUT
	i_xOverrideMode : BOOL;
END_VAR
VAR_OUTPUT
END_VAR
VAR

tonOvrd	:	TON;
tonDelOK : TON;
rtOK	:	R_TRIG;

END_VAR

(* This function block is different from the regular VRC in that CLOSING must be permitted. *)
(* Implemented for the funky valve 04 on LAMP *)
IF NOT iq_stValve.xOPN_OK and NOT tonOvrd.Q THEN
iq_stValve.pv_xOPN_SW := FALSE;
END_IF

(* Override logic *)
(* Goal: give ability to override, but do so in a way that people won't forget it.
Solution: Override only after ten seconds of override, protect against blips,
when the valve permission goes true for more than ten seconds consistently, remove override
*)

tonDelOK(IN:=iq_stValve.xOPN_OK, PT:=T#10S);
rtOK(CLK:=tonDelOK.Q);
IF rtOK.Q THEN iq_stValve.pv_xOvrdOpn :=FALSE; END_IF

//Override timer
tonOvrd(IN:=iq_stValve.pv_xOvrdOpn, PT:=T#10S);

(* Here's where the valve opens *)
iq_stValve.q_xOPN_DO := NOT iq_stValve.xCLS_OK OR ((iq_stValve.pv_xOPN_SW AND iq_stValve.xOPN_OK) OR (tonOvrd.Q AND i_xOverrideMode));

END_FUNCTION_BLOCK

// UnitTests/Functions/V_TO_INT
{attribute 'no_check'}
FUNCTION V_TO_INT : INT
VAR_INPUT
	analog : REAL;
END_VAR
VAR
	iBits :INT := 32767;
	iFullRange:INT := 10;
END_VAR

if ( iFullRange = 0 ) THEN iFullRange := 10;END_IF
V_TO_INT := REAL_TO_INT(analog * 32767 /iFullRange);

END_FUNCTION

// UnitTests/Gauges/FB_GCC_Test
FUNCTION_BLOCK FB_GCC_Test EXTENDS TcUnit.FB_TestSuite
VAR_INPUT
END_VAR
VAR_OUTPUT
END_VAR
VAR
	PG : ST_VG;
	fb_MKS422: FB_MKS422;
	//fb_MKS500: FB_MKS500;
	i_iPRESS_R AT %Q* :INT;
	cycle:INT :=0;
END_VAR

M_INIT();
M_Interlock();
M_CheckRange();
//M_SelfProtection();
cycle:=cycle+1;

METHOD M_CheckRange
VAR
	Expected:REAL;
	Actual:REAL;
	eStateExpected: E_PressureState;
	eStateActual: E_PressureState;
END_VAR
TEST('Check_Range');
Case This^.cycle of
	12:
	This^.i_iPRESS_R :=  V_TO_INT(0.61);
	This^.PG.rPRESS := 1E-4;
	This^.PG.xPRESS_OK := True;
	fb_MKS422.M_HVE(TRUE);
	
	15:
	TEST('MKS422_Range_937B');
	Expected :=1E-11 ;
	eStateExpected := Valid;
	Actual := This^.fb_MKS422.IG.rPRESS;
	eStateActual := This^.fb_MKS422.IG.eState;
	AssertTrue(This^.fb_MKS422.IG.xPRESS_OK, 'MKS422B xPRESS_OK is set to False');
	AssertEquals(eStateExpected,eStateActual,'MKS422B eState Fail');
	AssertEquals_REAL(Expected, Actual,1E-12, 'MKS422B rPress Fail');
	TEST_FINISHED_NAMED('MKS422_Range_937B');
	
	16:
	This^.i_iPRESS_R := V_TO_INT(2.4);
	This^.fb_MKS422.b937A:=TRUE;
	
	20:
	TEST('MKS422_Range_937A');
	Expected :=1E-8 ;
	Actual := This^.fb_MKS422.IG.rPRESS;
	eStateExpected := Valid;
	eStateActual := This^.fb_MKS422.IG.eState;
	AssertTrue(This^.fb_MKS422.IG.xPRESS_OK, 'MKS422A xPRESS_OK is set to False');
	AssertEquals(eStateExpected,eStateActual,'MKS422A eState Fail');
	AssertEquals_REAL(Expected, Actual,1E-9, 'MKS422A rPress Fail');
	TEST_FINISHED_NAMED('MKS422_Range_937A');

	
	21:
	This^.i_iPRESS_R :=  V_TO_INT(0.1);  
	
	
	24:
	TEST('MKS422_Range_Off');
	Expected :=0 ;
	eStateExpected := GaugeDisconnected;
	Actual := This^.fb_MKS422.IG.rPRESS;
	eStateActual := This^.fb_MKS422.IG.eState;
	AssertFalse(This^.fb_MKS422.IG.xPRESS_OK, 'MKS422A xPRESS_OK is set to True');
	AssertEquals(eStateExpected,eStateActual,'MKS422A eState Fail');
	AssertEquals_REAL(Expected, Actual,1, 'MKS422A rPress Fail');
	TEST_FINISHED_NAMED('MKS422_Range_Off');

	
	25:
	This^.i_iPRESS_R :=  V_TO_INT(10); 
	
	
	29:
	TEST('MKS422_Range_Invalid');
	Expected :=0 ;
	eStateExpected := PressInvalid;
	Actual := This^.fb_MKS422.IG.rPRESS;
	eStateActual := This^.fb_MKS422.IG.eState;
	AssertFalse(This^.fb_MKS422.IG.xPRESS_OK, 'MKS422A xPRESS_OK is set to True');
	AssertEquals(eStateExpected,eStateActual,'MKS422A eState Fail');
	AssertEquals_REAL(Expected, Actual,1, 'MKS422A rPress Fail');
	TEST_FINISHED_NAMED('MKS422_Range_Invalid');
	TEST_FINISHED_NAMED('Check_Range');

END_CASE

This^.fb_MKS422(PG:=This^.PG, IG=>);
END_METHOD

METHOD M_INIT
VAR
END_VAR
TEST('MKS422_Startup');
This^.PG.rPRESS := 1E-4;
This^.PG.xPRESS_OK := TRUE;
This^.fb_MKS422(PG:=This^.PG, IG=>);
IF( cycle = 3) THEN
	AssertFalse(This^.fb_MKS422.IG.xHV_SW, 'MKS422 xHV_SW set to True');
	AssertTrue(This^.fb_MKS422.IG.q_xHV_DIS, 'MKS422 q_xHV_DIS set to False');
	TEST_FINISHED_NAMED('MKS422_Startup');
End_IF;
END_METHOD

METHOD M_Interlock
VAR_INPUT
END_VAR
TEST('MKS422_Interlock_Active');
TEST('MKS422_Interlock_OK');
TEST('MKS422_Interlock_Lost');

Case cycle of
	1:
	This^.PG.rPRESS := 1E-1;
	This^.PG.xPRESS_OK := TRUE;
	fb_MKS422.M_HVE(TRUE);
	
	3:
	AssertFalse(This^.fb_MKS422.IG.xHV_SW, 'MKS422 xHV_SW set to True');
	AssertTrue(This^.fb_MKS422.IG.q_xHV_DIS, 'MKS422 q_xHV_DIS set to False');
	TEST_FINISHED_NAMED('MKS422_Interlock_Active');
	
	4:
	This^.PG.rPRESS := 1E-4;
	This^.PG.xPRESS_OK := True;
	fb_MKS422.M_HVE(TRUE);
	
	7:
	AssertTrue(This^.fb_MKS422.IG.xHV_SW, 'MKS422 xHV_SW set to False');
	AssertFalse(This^.fb_MKS422.IG.q_xHV_DIS, 'MKS422 q_xHV_DIS set to True');
	TEST_FINISHED_NAMED('MKS422_Interlock_OK');

	8:
	This^.PG.rPRESS := 1E-1;
	This^.PG.xPRESS_OK := False;
	This^.fb_MKS422(PG:=This^.PG, IG=>);
	
	11:
	AssertFalse(This^.fb_MKS422.IG.xHV_SW, 'MKS422 xHV_SW set to True');
	AssertTrue(This^.fb_MKS422.IG.q_xHV_DIS, 'MKS422 q_xHV_DIS set to False');
	TEST_FINISHED_NAMED('MKS422_Interlock_Lost');
END_CASE

This^.fb_MKS422(PG:=This^.PG, IG=>);
END_METHOD

METHOD M_SelfProtection
VAR_INPUT
END_VAR
// Switching the Cold cathode backon
TEST('MKS422_Interlock_OK_1');
This^.PG.rPRESS := 1E-4;
This^.PG.xPRESS_OK := True;
fb_MKS422.M_HVE(TRUE);
This^.fb_MKS422(PG:=This^.PG, IG=>);
AssertTrue(This^.fb_MKS422.IG.xHV_SW, 'MKS422 xHV_SW set to False');
AssertFalse(This^.fb_MKS422.IG.q_xHV_DIS, 'MKS422 q_xHV_DIS set to True');
TEST_FINISHED_NAMED('MKS422_Interlock_OK_1');

TEST('MKS422_Self_Protection');
This^.PG.rPRESS := 1E-3;
This^.PG.xPRESS_OK := TRUE;
This^.fb_MKS422(PG:=This^.PG, IG=>);
AssertFalse(This^.fb_MKS422.IG.xHV_SW, 'MKS422 xHV_SW set to True');
AssertTrue(This^.fb_MKS422.IG.q_xHV_DIS, 'MKS422 q_xHV_DIS set to False');
TEST_FINISHED_NAMED('MKS422_Self_Protection');
END_METHOD

END_FUNCTION_BLOCK

// UnitTests/Gauges/FB_GPI_Test
FUNCTION_BLOCK FB_GPI_Test EXTENDS TcUnit.FB_TestSuite
VAR_INPUT
END_VAR
VAR_OUTPUT
END_VAR
VAR
	fb_MKS275: FB_MKS275;
	fb_MKS317: FB_MKS317;
	i_iPRESS_R AT %Q* :INT;
	cycle:INT :=0;
END_VAR

M_INIT();
M_CheckRange();
cycle:=cycle+1;

METHOD M_CheckRange
VAR
	Expected:REAL;
	Actual:REAL;
	eStateExpected: E_PressureState;
	eStateActual: E_PressureState;
END_VAR

TEST('MKS275_Check_Range');
Case cycle of
	4:
	This^.i_iPRESS_R := V_TO_INT(3.674);
	Expected :=5 ;
	eStateExpected := Valid;
	
	7:
	TEST('MKS275_Range_R2');
	Actual := This^.fb_MKS275.PG.rPRESS;
	eStateActual := This^.fb_MKS275.PG.eState;
	AssertTrue(This^.fb_MKS275.PG.xPRESS_OK, 'MKS275 xPRESS_OK is set to False');
	AssertEquals(eStateExpected,eStateActual,'MKS275 eState Fail');
	AssertEquals_REAL(Expected, Actual,0.1, 'MKS275 rPress Fail');
	TEST_FINISHED_NAMED('MKS275_Range_R2');
	
	8:
	This^.i_iPRESS_R := V_TO_INT(5.614);
	Expected :=900 ;
	eStateExpected := Valid;
	
	
	12:
	TEST('MKS275_Range_R3');
	Actual := This^.fb_MKS275.PG.rPRESS;
	eStateActual := This^.fb_MKS275.PG.eState;
	AssertTrue(This^.fb_MKS275.PG.xPRESS_OK, 'MKS275 xPRESS_OK is set to False');
	AssertEquals(eStateExpected,eStateActual,'MKS275 eState Fail');
	AssertEquals_REAL(Expected, Actual,1, 'MKS275 rPress Fail');
	TEST_FINISHED_NAMED('MKS275_Range_R3');

	
	13:
	This^.i_iPRESS_R := V_TO_INT(0.3);
	Expected :=-1 ;
	eStateExpected := GaugeDisconnected;
	
	17:
	TEST('MKS275_Range_Off');
	Actual := This^.fb_MKS275.PG.rPRESS;
	eStateActual := This^.fb_MKS275.PG.eState;
	AssertTrue(This^.fb_MKS275.PG.xPRESS_OK, 'MKS275 xPRESS_OK is set to False');
	AssertEquals(eStateExpected,eStateActual,'MKS275 eState Fail');
	AssertEquals_REAL(Expected, Actual,1, 'MKS275 rPress Fail');
	TEST_FINISHED_NAMED('MKS275_Range_Off');

	
	18:
	This^.i_iPRESS_R := V_TO_INT(5.66);
	Expected :=-1 ;
	eStateExpected := OoR;
	
	22:
	TEST('MKS275_Range_OoR');
	Actual := This^.fb_MKS275.PG.rPRESS;
	eStateActual := This^.fb_MKS275.PG.eState;
	AssertTrue(This^.fb_MKS275.PG.xPRESS_OK, 'MKS275 xPRESS_OK is set to False');
	AssertEquals(eStateExpected,eStateActual,'MKS275 eState Fail');
	AssertEquals_REAL(Expected, Actual,1, 'MKS275 rPress Fail');
	TEST_FINISHED_NAMED('MKS275_Range_OoR');
	TEST_FINISHED_NAMED('MKS275_Check_Range');
	
END_CASE

This^.fb_MKS275(PG=>);
This^.fb_MKS317(PG=>);
END_METHOD

METHOD M_INIT
VAR
	Expected:REAL;
	Actual:REAL;
	eStateExpected: E_PressureState;
	eStateActual: E_PressureState;
END_VAR
// Start the Test
TEST('MKS275_Startup');
//Assign Voltage to FB
This^.i_iPRESS_R := V_TO_INT(0.384);
// Assigne expected result corresponing to the test input
Expected :=0.001 ;
eStateExpected := Valid;
//Instantiate the function block
This^.fb_MKS275(PG=>);
// Wait for few cycles 
IF( cycle = 3) THEN
	// Check the results
	Actual := This^.fb_MKS275.PG.rPRESS;
	eStateActual := This^.fb_MKS275.PG.eState;
	AssertTrue(This^.fb_MKS275.PG.xPRESS_OK, 'MKS275 xPRESS_OK is set to False');
	AssertEquals(eStateExpected,eStateActual,'MKS275 eState Fail');
	AssertEquals_REAL(Expected, Actual,0.0001, 'MKS275 rPress Fail');
	TEST_FINISHED_NAMED('MKS275_Startup');
END_IF
END_METHOD

END_FUNCTION_BLOCK

// UnitTests/Pumps/FB_PIP_Test
FUNCTION_BLOCK FB_PIP_Test EXTENDS TcUnit.FB_TestSuite
VAR_INPUT
END_VAR
VAR_OUTPUT
END_VAR
VAR
	PG : ST_VG;
	fb_PIP_GAMMA: FB_PIP_GAMMA;
END_VAR

M_INIT();
M_Interlock();
M_AutoStart();

METHOD M_AutoStart
VAR_INPUT
END_VAR
TEST('PIP_Auto_Restart');
This^.PG.rPRESS := 1E-6;
This^.PG.xPRESS_OK := TRUE;
This^.fb_PIP_GAMMA(i_stGauge:=PG, stPump=>, q_IG=>);
AssertTrue(This^.fb_PIP_GAMMA.stPump.q_xHVEna_DO, 'PIP HVEna_DO set to false');
TEST_FINISHED_NAMED('PIP_Auto_Restart');
END_METHOD

METHOD M_Check_State
VAR_INPUT
END_VAR
END_METHOD

METHOD M_INIT
VAR_INPUT
END_VAR
TEST('PIP_Startup');
This^.PG.rPRESS := 1E-1;
This^.PG.xPRESS_OK := TRUE;
This^.fb_PIP_GAMMA(i_stGauge:=PG, stPump=>, q_IG=>);
AssertFalse(This^.fb_PIP_GAMMA.stPump.xHVEna_SW, 'PIP xHVEna_SW set to True');
AssertFalse(This^.fb_PIP_GAMMA.stPump.q_xHVEna_DO, 'PIP HVEna_DO set to True');
TEST_FINISHED_NAMED('PIP_Startup');
END_METHOD

METHOD M_Interlock
VAR_INPUT
END_VAR
TEST('PIP_Interlock_Active');
This^.PG.rPRESS := 1E-1;
This^.PG.xPRESS_OK := True;
This^.fb_PIP_GAMMA.M_Run(TRUE);
This^.fb_PIP_GAMMA(i_stGauge:=PG, stPump=>, q_IG=>);
AssertFalse(This^.fb_PIP_GAMMA.stPump.xHVEna_SW, 'PIP xHVEna_SW set to True');
AssertFalse(This^.fb_PIP_GAMMA.stPump.q_xHVEna_DO, 'PIP HVEna_DO set to True');
TEST_FINISHED_NAMED('PIP_Interlock_Active');

TEST('PIP_Interlock_OK');
This^.PG.rPRESS := 1E-9;
This^.PG.xPRESS_OK := True;
This^.fb_PIP_GAMMA.M_Run(TRUE);
This^.fb_PIP_GAMMA(i_stGauge:=PG, stPump=>, q_IG=>);
AssertTrue(This^.fb_PIP_GAMMA.stPump.xHVEna_SW, 'PIP xHVEna_SW set to False');
AssertTrue(This^.fb_PIP_GAMMA.stPump.q_xHVEna_DO, 'PIP HVEna_DO set to False');
TEST_FINISHED_NAMED('PIP_Interlock_OK');

TEST('PIP_Interlock_Lost');
This^.PG.rPRESS := 1E-9;
This^.PG.xPRESS_OK := False;
This^.fb_PIP_GAMMA(i_stGauge:=PG, stPump=>, q_IG=>);
AssertFalse(This^.fb_PIP_GAMMA.stPump.xHVEna_SW, 'PIP xHVEna_SW set to True');
AssertFalse(This^.fb_PIP_GAMMA.stPump.q_xHVEna_DO, 'PIP HVEna_DO set to True');
TEST_FINISHED_NAMED('PIP_Interlock_Lost');
END_METHOD

END_FUNCTION_BLOCK

// UnitTests/Pumps/FB_PTM_Test
FUNCTION_BLOCK FB_PTM_Test EXTENDS TcUnit.FB_TestSuite
VAR_INPUT
END_VAR
VAR_OUTPUT
END_VAR
VAR
	fb_TwisTorr: FB_PTM_TwisTorr;
	fb_PTM_Ebara_010M:FB_PTM_Ebara_010M;
	
	cycle:INT :=0;
	(*IO*)
	q_iSpeedSet AT %I* :INT;
	i_diCurSpd AT %Q* :INT;
	
	i_iRawSpeed AT %Q* : INT; // Link to Analog input
	i_iTempMon AT %Q* : INT; // Link to Analog input -- input Voltage according to the pump temprature 0->5V 0->100C
	i_iCurrentMon AT %Q* : INT; //Link to Analog -- input Voltage to the output current of motor 0->5V 0->10A
	
END_VAR

M_INIT();
M_Interlock();
M_PTM_EBARA();
cycle:=cycle+1;

METHOD M_INIT : BOOL
VAR_INPUT
END_VAR
TEST('PTM_Twistorr_Startup');
fb_TwisTorr(i_xExtILKOk:= TRUE , iq_stPtm=> );
IF( cycle = 3) THEN
	AssertFalse(fb_TwisTorr.iq_stPtm.xRunSW ,'PTM Twistorr xRunSW is set to true');	
	AssertFalse(fb_TwisTorr.iq_stPtm.q_RunDO ,'PTM Twistorr q_RunDO is set to true');
	TEST_FINISHED_NAMED('PTM_Twistorr_Startup');
END_IF


TEST('PTM_Ebara011M_Startup');
fb_PTM_Ebara_010M(i_xExtILKOk:= TRUE , iq_stPtm=> );
IF( cycle = 3) THEN
	AssertFalse(fb_PTM_Ebara_010M.iq_stPtm.xRunSW ,'PTM Ebara011M xRunSW is set to true');	
	AssertFalse(fb_PTM_Ebara_010M.iq_stPtm.q_RunDO ,'PTM Ebara011M q_RunDO is set to true');
	AssertFalse(fb_PTM_Ebara_010M.iq_stPtm.q_xProtection ,'PTM Ebara011M q_xProtection is set to True');
	TEST_FINISHED_NAMED('PTM_Ebara011M_Startup');
END_IF
END_METHOD

METHOD M_Interlock
VAR_INPUT
END_VAR
TEST('PTM_Twistorr_Interlock_Active');
fb_TwisTorr.M_Run(TRUE);
fb_TwisTorr(i_xExtILKOk:= FALSE , iq_stPtm=> );
IF( cycle = 3) THEN
	AssertFalse(fb_TwisTorr.iq_stPtm.xRunSW ,'PTM Twistorr xRunSW is set to true');	
	AssertFalse(fb_TwisTorr.iq_stPtm.q_RunDO ,'PTM Twistorr q_RunDO is set to true');
	TEST_FINISHED_NAMED('PTM_Twistorr_Interlock_Active');
END_IF

TEST('PTM_Twistorr_Interlock_OK');
fb_TwisTorr.M_Run(TRUE);
fb_TwisTorr(i_xExtILKOk:= TRUE , iq_stPtm=> );
IF( cycle = 3) THEN
	AssertTrue(fb_TwisTorr.iq_stPtm.xRunSW ,'PTM Twistorr xRunSW is set to False');	
	AssertTrue(fb_TwisTorr.iq_stPtm.q_RunDO ,'PTM Twistorr q_RunDO is set to False');
	TEST_FINISHED_NAMED('PTM_Twistorr_Interlock_OK');
END_IF

TEST('PTM_Twistorr_Interlock_Lost');
fb_TwisTorr(i_xExtILKOk:= FALSE , iq_stPtm=> );
IF( cycle = 3) THEN
	AssertFalse(fb_TwisTorr.iq_stPtm.xRunSW ,'PTM Twistorr xRunSW is set to true');	
	AssertFalse(fb_TwisTorr.iq_stPtm.q_RunDO ,'PTM Twistorr q_RunDO is set to true');
	TEST_FINISHED_NAMED('PTM_Twistorr_Interlock_Lost');
END_IF
END_METHOD

METHOD M_PTM_EBARA
VAR
	Expected:REAL;
	Actual:REAL;
	diExpected:DINT;
	diActual: DINT;
END_VAR
TEST('PTM_EBARA_AI');
This^.i_iRawSpeed := v_to_int(5);
This^.i_iTempMon := v_to_int(2.5);
THIS^.i_iCurrentMon := v_to_int(2.5);
//THIS^.q_iSpeedSet := 560;

fb_PTM_Ebara_010M(
	i_xExtILKOk:= TRUE , 
	i_rMaxBackingPressure:= 1, 
	iq_stPTM=> );


IF( cycle = 10) THEN
	Expected := 5;
	Actual := (fb_PTM_Ebara_010M.iq_stPTM.i_rCurrentMon);
	AssertEquals_REAL(Expected, Actual,0.1, 'PTM EBARA010 i_iCurrentMon Fail');
	Expected := 50;
	Actual := (fb_PTM_Ebara_010M.iq_stPTM.i_rTempMon);
	AssertEquals_REAL(Expected, Actual,0.1, 'PTM EBARA010 i_iTempMon Fail');
	diExpected := 0;
	diActual := fb_PTM_Ebara_010M.iq_stPTM.q_iSpeedSet;
	AssertEquals(diExpected, diActual, 'PTM EBARA010 q_iSpeedSet Fail');
	diExpected := 560;
	diActual :=  fb_PTM_Ebara_010M.iq_stPTM.i_diCurSpd;
	AssertEquals(diExpected, diActual, 'PTM EBARA010 i_diCurSpd Fail');
	TEST_FINISHED_NAMED('PTM_EBARA_AI');
	
	
End_IF;
END_METHOD

END_FUNCTION_BLOCK

// UnitTests/Valves/FB_VGC_Test
FUNCTION_BLOCK FB_VGC_Test EXTENDS TcUnit.FB_TestSuite
VAR_INPUT
END_VAR
VAR_OUTPUT
END_VAR
VAR
	VGC: FB_VGC;
	US_IG : ST_VG;
	DS_IG : ST_VG;
	io_fbFFHWO    :    FB_HardwareFFOutput;
	TotalTests : INT:=0;
	ex               : __SYSTEM.ExceptionCode;
END_VAR

M_INIT();
M_Interlock();

METHOD M_Check_State
VAR_INPUT
END_VAR
END_METHOD

METHOD M_INIT : BOOL
VAR//_INPUT
	
END_VAR
TEST('VGC_Startup');
This^.US_IG.rPRESS := 1E-9;
This^.US_IG.xPRESS_OK := TRUE;
This^.US_IG.xAT_VAC := TRUE;

This^.DS_IG.rPRESS := 1E-9;
This^.DS_IG.xPRESS_OK := TRUE;

(*This^.VGC(
	i_stUSG:= This^.US_IG, 
	i_stDSG:= This^.DS_IG , 
	i_xDis_DPIlk:= FALSE, 
	i_xEPS_OK:= TRUE , 
	//i_xPMPS_OK:= TRUE, 
	i_xExt_OK:= TRUE, 
	i_xOverrideMode:= , 
	i_xReset:= , 
	iq_stValve=> , 
	xMPS_OK=> , 
	io_fbFFHWO:= This^.io_fbFFHWO,
	fbArbiter:=g_fbArbiter);
*)
AssertFalse(This^.VGC.iq_stValve.pv_xOPN_SW,'VGC pv_xOPN_SW is set to true');
AssertFalse(VGC.iq_stValve.q_xOPN_DO,'VGC q_xOPN_DO is set to true');
TEST_FINISHED_NAMED('VGC_Startup');
END_METHOD

METHOD M_Interlock : BOOL
VAR//_INPUT
	
END_VAR
// Test interlock is active and attempting to open valve
TEST('VGC_Interlock_Active');
This^.US_IG.xPRESS_OK := FALSE; 
This^.DS_IG.xPRESS_OK := FALSE;
VGC.M_Set_OPN_SW(TRUE);
// run the function block one more time
(*VGC(
	i_stUSG:= US_IG, 
	i_stDSG:= DS_IG , 
	i_xDis_DPIlk:= FALSE, 
	i_xEPS_OK:= TRUE , 
	i_xPMPS_OK:= TRUE , 
	i_xExt_OK:= TRUE, 
	i_xOverrideMode:= , 
	i_xReset:= , 
	iq_stValve=> , 
	xMPS_OK=> , 
	io_fbFFHWO:= io_fbFFHWO);*)
AssertFalse(VGC.iq_stValve.pv_xOPN_SW,'VGC pv_xOPN_SW is set to true');
AssertFalse(VGC.iq_stValve.q_xOPN_DO,'VGC q_xOPN_DO is set to true');
TEST_FINISHED_NAMED('VGC_Interlock_Active');
// Test interlock is not active and attempting to open valve
TEST('VGC_Interlock_OK');
This^.US_IG.xPRESS_OK := TRUE; 
This^.DS_IG.xPRESS_OK := TRUE;
VGC.M_Set_OPN_SW(TRUE);
// run the function block one more time
(*VGC(
	i_stUSG:= US_IG, 
	i_stDSG:= DS_IG , 
	i_xDis_DPIlk:= FALSE, 
	i_xEPS_OK:= , 
	i_xPMPS_OK:= , 
	i_xExt_OK:= , 
	i_xOverrideMode:= , 
	i_xReset:= , 
	iq_stValve=> , 
	xMPS_OK=> , 
	io_fbFFHWO:= io_fbFFHWO);*)
AssertTrue(VGC.iq_stValve.pv_xOPN_SW,'VGC pv_xOPN_SW is set to false');
AssertTrue(VGC.iq_stValve.q_xOPN_DO,'VGC q_xOPN_DO is set to false');
TEST_FINISHED_NAMED('VGC_Interlock_OK');
// Test interlock ok lost while valve is open
TEST('VGC_Interlock_Lost');
This^.US_IG.xPRESS_OK := False; 
This^.DS_IG.xPRESS_OK := TRUE;
// run the function block one more time
(*VGC(
	i_stUSG:= US_IG, 
	i_stDSG:= DS_IG , 
	i_xDis_DPIlk:= FALSE, 
	i_xEPS_OK:= , 
	i_xPMPS_OK:= , 
	i_xExt_OK:= , 
	i_xOverrideMode:= , 
	i_xReset:= , 
	iq_stValve=> , 
	xMPS_OK=> , 
	io_fbFFHWO:= io_fbFFHWO);*)
AssertFalse(VGC.iq_stValve.pv_xOPN_SW,'VGC pv_xOPN_SW is set to true');
AssertFalse(VGC.iq_stValve.q_xOPN_DO,'VGC q_xOPN_DO is set to true');
TEST_FINISHED_NAMED('VGC_Interlock_Lost');
END_METHOD

END_FUNCTION_BLOCK

// UnitTests/Valves/FB_VRC_Test
FUNCTION_BLOCK FB_VRC_Test EXTENDS TcUnit.FB_TestSuite
VAR_INPUT
END_VAR
VAR_OUTPUT
END_VAR
VAR
	VRC: FB_VRC;
	ex               : __SYSTEM.ExceptionCode;
END_VAR

M_INIT();
M_Interlock();

METHOD M_Check_State
VAR_INPUT
END_VAR
END_METHOD

METHOD M_INIT : BOOL
VAR//_INPUT
	
	
	Interlock_OK :BOOL := TRUE;
 
	ex: INT;
END_VAR
TEST('VRC_Startup');
//__TRY
VRC(i_xExtILK_OK:= Interlock_OK, i_xOverrideMode:= , iq_stValve=> );
AssertFalse(VRC.iq_stValve.q_xOPN_DO,'VRC q_xOPN_DO is set to true');
AssertFalse(VRC.iq_stValve.pv_xOPN_SW,'VRC pv_xOPN_SW is set to true');
//__CATCH(ex) 
//__FINALLY
TEST_FINISHED_NAMED('VRC_Startup');
//__ENDTRY
END_METHOD

METHOD M_Interlock
VAR
	US_IG : ST_VG;
	DS_IG : ST_VG;
	
	VRC: FB_VRC;
END_VAR
TEST('VRC_Interlock_Active');
VRC.M_Set_OPN_SW (TRUE);
VRC(i_xExtILK_OK:= FALSE, i_xOverrideMode:= , iq_stValve=> );
AssertFalse(VRC.iq_stValve.pv_xOPN_SW,'VRC open_SW is set to true');
AssertFalse(VRC.iq_stValve.q_xOPN_DO,'VRC open DO is set to true');
TEST_FINISHED_NAMED('VRC_Interlock_Active');

TEST('VRC_Interlock_OK');
VRC.M_Set_OPN_SW (TRUE);
VRC(i_xExtILK_OK:= TRUE, i_xOverrideMode:= , iq_stValve=> );
AssertTrue(VRC.iq_stValve.pv_xOPN_SW,'VRC open_SW is set to FALSE');
AssertTrue(VRC.iq_stValve.q_xOPN_DO,'VRC open DO is set to FALSE');
TEST_FINISHED_NAMED('VRC_Interlock_OK');

TEST('VRC_Interlock_Lost');
VRC(i_xExtILK_OK:= FALSE, i_xOverrideMode:= , iq_stValve=> );
AssertFalse(VRC.iq_stValve.pv_xOPN_SW,'VRC open_SW is set to true');
AssertFalse(VRC.iq_stValve.q_xOPN_DO,'VRC open DO is set to true');
TEST_FINISHED_NAMED('VRC_Interlock_Lost');
END_METHOD

END_FUNCTION_BLOCK

// UnitTests/PRG_Test
PROGRAM PRG_Test
VAR
	fb_VGC_Test: FB_VGC_Test;
	fb_VRC_Test: FB_VRC_Test;
	fb_PIP_Test: FB_PIP_Test;
	fb_PTM_Test: FB_PTM_Test;
	fb_GPI_Test:FB_GPI_Test;
	fb_GCC_Test:FB_GCC_Test;

	TotalTests : INT:=0;
END_VAR


TcUnit.RUN();

END_PROGRAM
